// TIA Portal V17 export
// export: Created 2022-06-16T09:21:08.2779505Z, ExportSetting WithDefaults, DisplayName Totally Integrated Automation Portal, DisplayVersion V17, DisplayName TIA Portal Openness, DisplayVersion V17, DisplayName TIA Portal Version Control Interface, DisplayVersion V17, DisplayName STEP 7 Professional, DisplayVersion V17, DisplayName STEP 7 Safety, DisplayVersion V17, DisplayName WinCC Advanced, DisplayVersion V17
TYPE "typeMoveStatus"
// stored: IsFailsafeCompliant false
   STRUCT
      global : Bool;
      axis : Array[1.."AXIS_NUM"] of Bool;
   END_STRUCT;
END_TYPE
